{attribute 'linkalways'} 
{attribute 'no_explicit_call' := 'This FB is a CLASS and must be accessed using methods or properties'}
{attribute 'enable_dynamic_creation'}
FUNCTION_BLOCK AliasDatatypeAddedEvent EXTENDS Disposable IMPLEMENTS I_AliasDatatypeAddedEvent
VAR
	_target : I_AliasDatatype;
END_VAR

METHOD FB_init : BOOL
VAR_INPUT
	bInitRetains : BOOL; // if TRUE, the retain variables are initialized (warm start / cold start)
	bInCopyCode : BOOL;  // if TRUE, the instance afterwards gets moved into the copy code (online change)
	Target : I_AliasDatatype;
END_VAR
This^._target := Target;
END_METHOD

PROPERTY PUBLIC Target : I_AliasDatatype
GET
Target := _target;
END_GET
END_PROPERTY

END_FUNCTION_BLOCK

(* stored: Version 1.1.0.1, ProductVersion 3.1.4024.12
   POU AliasDatatypeAddedEvent: Id {451a3ea1-7720-0619-0ec0-706f7dfcaae2}, SpecialFunc None
   Folder Constructor: Id {317f6278-4a13-088d-1323-409cab9ac564}
   Method FB_init: Id {59c764d9-7941-0033-0ffc-f45acd7d9e24}
   Property Target: Id {0467fab9-db87-08fc-17fa-c29fea0aaf24}
   Get Get: Id {b78cada4-ce57-0420-339d-1c28b593e944} *)
